LIN {X 0,Y 128.557,Z 1225.64,A -85,B 0,C 180,E1 5972.035,E2 5972.035} C_VEL
LIN {X 0,Y 143.599,Z 1214.931,A -85,B 0,C 180,E1 5965.157,E2 5965.157} C_VEL
LIN {X 0,Y 159.546,Z 1202.831,A -85,B 0,C 180,E1 5959.947,E2 5959.947} C_VEL
LIN {X 0,Y 175.745,Z 1189.232,A -85,B 0,C 180,E1 5955.959,E2 5955.959} C_VEL
LIN {X 0,Y 191.807,Z 1174.321,A -85,B 0,C 180,E1 5952.898,E2 5952.898} C_VEL
LIN {X 0,Y 207.044,Z 1158.532,A -85,B 0,C 180,E1 5950.574,E2 5950.574} C_VEL
LIN {X 0,Y 221.552,Z 1141.458,A -85,B 0,C 180,E1 5948.77,E2 5948.77} C_VEL
LIN {X 0,Y 234.912,Z 1123.521,A -85,B 0,C 180,E1 5947.392,E2 5947.392} C_VEL
LIN {X 0,Y 247.459,Z 1104.198,A -85,B 0,C 180,E1 5946.316,E2 5946.316} C_VEL
LIN {X 0,Y 258.166,Z 1084.964,A -85,B 0,C 180,E1 5945.551,E2 5945.551} C_VEL
LIN {X 0,Y 267.457,Z 1065.024,A -85,B 0,C 180,E1 5944.964,E2 5944.964} C_VEL
LIN {X 0,Y 275.777,Z 1043.211,A -85,B 0,C 180,E1 5944.432,E2 5944.432} C_VEL
LIN {X 0,Y 282.412,Z 1020.924,A -85,B 0,C 180,E1 5943.975,E2 5943.975} C_VEL
LIN {X 0,Y 287.197,Z 998.303,A -85,B 0,C 180,E1 5943.578,E2 5943.578} C_VEL
LIN {X 0,Y 291.386,Z 967,A -85,B 0,C 180,E1 5943.086,E2 5943.086} C_VEL
LIN {X 0,Y 296.698,Z 921.737,A -85,B 0,C 180,E1 5942.366,E2 5942.366} C_VEL
LIN {X 0,Y 296.244,Z 920.618,A -85,B 0,C 180,E1 5938.452,E2 5938.452} C_VEL
LIN {X 0,Y 296.574,Z 921.627,A -85,B 0,C 180,E1 5935.555,E2 5935.555} C_VEL
LIN {X 0,Y 290.553,Z 972.951,A -85,B 0,C 180,E1 5934.658,E2 5934.658} C_VEL
LIN {X 0,Y 287.245,Z 994.55,A -85,B 0,C 180,E1 5934.116,E2 5934.116} C_VEL
LIN {X 0,Y 282.043,Z 1017.129,A -85,B 0,C 180,E1 5933.394,E2 5933.394} C_VEL
LIN {X 0,Y 275.76,Z 1037.409,A -85,B 0,C 180,E1 5932.582,E2 5932.582} C_VEL
LIN {X 0,Y 267.826,Z 1057.375,A -85,B 0,C 180,E1 5931.603,E2 5931.603} C_VEL
LIN {X 0,Y 258.412,Z 1076.786,A -85,B 0,C 180,E1 5930.422,E2 5930.422} C_VEL
LIN {X 0,Y 248.14,Z 1094.686,A -85,B 0,C 180,E1 5929.083,E2 5929.083} C_VEL
LIN {X 0,Y 236.579,Z 1111.772,A -85,B 0,C 180,E1 5927.488,E2 5927.488} C_VEL
LIN {X 0,Y 224,Z 1127.849,A -85,B 0,C 180,E1 5925.599,E2 5925.599} C_VEL
LIN {X 0,Y 210.772,Z 1142.685,A -85,B 0,C 180,E1 5923.378,E2 5923.378} C_VEL
LIN {X 0,Y 196.129,Z 1156.912,A -85,B 0,C 180,E1 5920.577,E2 5920.577} C_VEL
LIN {X 0,Y 181.129,Z 1169.686,A -85,B 0,C 180,E1 5917.196,E2 5917.196} C_VEL
LIN {X 0,Y 165.996,Z 1181.07,A -85,B 0,C 180,E1 5913.054,E2 5913.054} C_VEL
LIN {X 0,Y 151.049,Z 1191.002,A -85,B 0,C 180,E1 5907.915,E2 5907.915} C_VEL
LIN {X 0,Y 136.729,Z 1199.368,A -85,B 0,C 180,E1 5901.484,E2 5901.484} C_VEL
LIN {X 0,Y 123.709,Z 1206.226,A -85,B 0,C 180,E1 5893.391,E2 5893.391} C_VEL
LIN {X 0,Y 113.281,Z 1211.302,A -85,B 0,C 180,E1 5883.783,E2 5883.783} C_VEL
LIN {X 0,Y 105.924,Z 1214.694,A -85,B 0,C 180,E1 5872.768,E2 5872.768} C_VEL
LIN {X 0,Y 102.021,Z 1216.463,A -85,B 0,C 180,E1 5861.303,E2 5861.303} C_VEL
LIN {X 0,Y 100.923,Z 1217.057,A -85,B 0,C 180,E1 5850.568,E2 5850.568} C_VEL
LIN {X 0,Y 101.896,Z 1216.542,A -85,B 0,C 180,E1 5839.255,E2 5839.255} C_VEL
LIN {X 0,Y 105.398,Z 1214.996,A -85,B 0,C 180,E1 5828.287,E2 5828.287} C_VEL
LIN {X 0,Y 112.423,Z 1211.729,A -85,B 0,C 180,E1 5817.146,E2 5817.146} C_VEL
LIN {X 0,Y 123.108,Z 1206.598,A -85,B 0,C 180,E1 5806.984,E2 5806.984} C_VEL
LIN {X 0,Y 135.387,Z 1200.239,A -85,B 0,C 180,E1 5799.157,E2 5799.157} C_VEL
LIN {X 0,Y 149.543,Z 1192.037,A -85,B 0,C 180,E1 5792.603,E2 5792.603} C_VEL
LIN {X 0,Y 164.371,Z 1182.32,A -85,B 0,C 180,E1 5787.367,E2 5787.367} C_VEL
LIN {X 0,Y 180.239,Z 1170.572,A -85,B 0,C 180,E1 5782.951,E2 5782.951} C_VEL
LIN {X 0,Y 195.213,Z 1157.984,A -85,B 0,C 180,E1 5779.542,E2 5779.542} C_VEL
LIN {X 0,Y 209.83,Z 1143.86,A -85,B 0,C 180,E1 5776.714,E2 5776.714} C_VEL
LIN {X 0,Y 223.492,Z 1128.733,A -85,B 0,C 180,E1 5774.409,E2 5774.409} C_VEL
LIN {X 0,Y 236.522,Z 1112.193,A -85,B 0,C 180,E1 5772.45,E2 5772.45} C_VEL
LIN {X 0,Y 248.371,Z 1094.704,A -85,B 0,C 180,E1 5770.817,E2 5770.817} C_VEL
LIN {X 0,Y 258.962,Z 1076.211,A -85,B 0,C 180,E1 5769.439,E2 5769.439} C_VEL
LIN {X 0,Y 268.715,Z 1055.867,A -85,B 0,C 180,E1 5768.22,E2 5768.22} C_VEL
LIN {X 0,Y 276.379,Z 1036.383,A -85,B 0,C 180,E1 5767.275,E2 5767.275} C_VEL
LIN {X 0,Y 282.83,Z 1015.172,A -85,B 0,C 180,E1 5766.44,E2 5766.44} C_VEL
LIN {X 0,Y 287.696,Z 993.438,A -85,B 0,C 180,E1 5765.758,E2 5765.758} C_VEL
LIN {X 0,Y 291.067,Z 970.64,A -85,B 0,C 180,E1 5765.196,E2 5765.196} C_VEL
LIN {X 0,Y 296.81,Z 921.706,A -85,B 0,C 180,E1 5764.329,E2 5764.329} C_VEL
LIN {X 0,Y 296.476,Z 920.939,A -85,B 0,C 180,E1 5760.773,E2 5760.773} C_VEL
LIN {X 0,Y 296.913,Z 922.137,A -85,B 0,C 180,E1 5757.598,E2 5757.598} C_VEL
LIN {X 0,Y 288.086,Z 994.765,A -85,B 0,C 180,E1 5756.486,E2 5756.486} C_VEL
LIN {X 0,Y 283.454,Z 1017.452,A -85,B 0,C 180,E1 5756.093,E2 5756.093} C_VEL
LIN {X 0,Y 277.274,Z 1039.329,A -85,B 0,C 180,E1 5755.657,E2 5755.657} C_VEL
LIN {X 0,Y 269.907,Z 1059.813,A -85,B 0,C 180,E1 5755.182,E2 5755.182} C_VEL
LIN {X 0,Y 260.611,Z 1080.49,A -85,B 0,C 180,E1 5754.602,E2 5754.602} C_VEL
LIN {X 0,Y 249.889,Z 1100.411,A -85,B 0,C 180,E1 5753.864,E2 5753.864} C_VEL
LIN {X 0,Y 238.282,Z 1118.997,A -85,B 0,C 180,E1 5752.908,E2 5752.908} C_VEL
LIN {X 0,Y 225.356,Z 1136.862,A -85,B 0,C 180,E1 5751.64,E2 5751.64} C_VEL
LIN {X 0,Y 210.819,Z 1154.455,A -85,B 0,C 180,E1 5749.924,E2 5749.924} C_VEL
LIN {X 0,Y 205.526,Z 1160.022,A -85,B 0,C 180,E1 5749.522,E2 5749.522} C_VEL
LIN {X 0,Y 190.415,Z 1173.211,A -85,B 0,C 180,E1 5749.253,E2 5749.253} C_VEL
LIN {X 0,Y 184.72,Z 1178.127,A -85,B 0,C 180,E1 5748.684,E2 5748.684} C_VEL
LIN {X 0,Y 168.259,Z 1192.432,A -85,B 0,C 180,E1 5745.598,E2 5745.598} C_VEL
LIN {X 0,Y 151.713,Z 1205.274,A -85,B 0,C 180,E1 5741.559,E2 5741.559} C_VEL
LIN {X 0,Y 134.693,Z 1217.324,A -85,B 0,C 180,E1 5735.904,E2 5735.904} C_VEL
LIN {X 0,Y 119.422,Z 1227.418,A -85,B 0,C 180,E1 5728.646,E2 5728.646} C_VEL
LIN {X 0,Y 106.632,Z 1235.615,A -85,B 0,C 180,E1 5719.419,E2 5719.419} C_VEL
LIN {X 0,Y 96.869,Z 1242.354,A -85,B 0,C 180,E1 5707.515,E2 5707.515} C_VEL
LIN {X 0,Y 91.73,Z 1247.309,A -85,B 0,C 180,E1 5693.784,E2 5693.784} C_VEL
LIN {X 0,Y 91.202,Z 1250.049,A -85,B 0,C 180,E1 5681.381,E2 5681.381} C_VEL
LIN {X 0,Y 92.698,Z 1251.177,A -85,B 0,C 180,E1 5671.854,E2 5671.854} C_VEL
LIN {X 0,Y 92.812,Z 1251.22,A -85,B 0,C 180,E1 5668.765,E2 5668.765} C_VEL
LIN {X 0,Y 91.266,Z 1250.151,A -85,B 0,C 180,E1 5659.267,E2 5659.267} C_VEL
LIN {X 0,Y 91.617,Z 1247.454,A -85,B 0,C 180,E1 5646.867,E2 5646.867} C_VEL
LIN {X 0,Y 96.53,Z 1242.58,A -85,B 0,C 180,E1 5633.077,E2 5633.077} C_VEL
LIN {X 0,Y 106.097,Z 1235.924,A -85,B 0,C 180,E1 5621.071,E2 5621.071} C_VEL
LIN {X 0,Y 118.748,Z 1227.765,A -85,B 0,C 180,E1 5611.746,E2 5611.746} C_VEL
LIN {X 0,Y 133.936,Z 1217.741,A -85,B 0,C 180,E1 5604.394,E2 5604.394} C_VEL
LIN {X 0,Y 150.911,Z 1205.757,A -85,B 0,C 180,E1 5598.663,E2 5598.663} C_VEL
LIN {X 0,Y 167.368,Z 1193.045,A -85,B 0,C 180,E1 5594.588,E2 5594.588} C_VEL
LIN {X 0,Y 183.649,Z 1178.921,A -85,B 0,C 180,E1 5591.489,E2 5591.489} C_VEL
LIN {X 0,Y 199.951,Z 1163.067,A -85,B 0,C 180,E1 5589.043,E2 5589.043} C_VEL
LIN {X 0,Y 214.685,Z 1146.942,A -85,B 0,C 180,E1 5587.261,E2 5587.261} C_VEL
LIN {X 0,Y 228.659,Z 1129.463,A -85,B 0,C 180,E1 5585.87,E2 5585.87} C_VEL
LIN {X 0,Y 241.398,Z 1111.157,A -85,B 0,C 180,E1 5584.82,E2 5584.82} C_VEL
LIN {X 0,Y 252.588,Z 1092.7,A -85,B 0,C 180,E1 5584.052,E2 5584.052} C_VEL
LIN {X 0,Y 262.931,Z 1072.464,A -85,B 0,C 180,E1 5583.45,E2 5583.45} C_VEL
LIN {X 0,Y 271.757,Z 1051.492,A -85,B 0,C 180,E1 5582.952,E2 5582.952} C_VEL
LIN {X 0,Y 279.127,Z 1029.628,A -85,B 0,C 180,E1 5582.514,E2 5582.514} C_VEL
LIN {X 0,Y 284.822,Z 1007.269,A -85,B 0,C 180,E1 5582.125,E2 5582.125} C_VEL
LIN {X 0,Y 288.68,Z 984.724,A -85,B 0,C 180,E1 5581.774,E2 5581.774} C_VEL
LIN {X 0,Y 295.41,Z 929.134,A -85,B 0,C 180,E1 5580.921,E2 5580.921} C_VEL
LIN {X 0,Y 295.275,Z 928.654,A -85,B 0,C 180,E1 5578.059,E2 5578.059} C_VEL
LIN {X 0,Y 295.326,Z 929.178,A -85,B 0,C 180,E1 5576.997,E2 5576.997} C_VEL
LIN {X 0,Y 289.639,Z 976.58,A -85,B 0,C 180,E1 5576.161,E2 5576.161} C_VEL
LIN {X 0,Y 286.245,Z 997.561,A -85,B 0,C 180,E1 5575.639,E2 5575.639} C_VEL
LIN {X 0,Y 281.067,Z 1019.164,A -85,B 0,C 180,E1 5574.966,E2 5574.966} C_VEL
LIN {X 0,Y 274.378,Z 1040.054,A -85,B 0,C 180,E1 5574.157,E2 5574.157} C_VEL
LIN {X 0,Y 266.317,Z 1059.866,A -85,B 0,C 180,E1 5573.22,E2 5573.22} C_VEL
LIN {X 0,Y 256.885,Z 1078.796,A -85,B 0,C 180,E1 5572.114,E2 5572.114} C_VEL
LIN {X 0,Y 246.122,Z 1097.056,A -85,B 0,C 180,E1 5570.803,E2 5570.803} C_VEL
LIN {X 0,Y 234.074,Z 1114.446,A -85,B 0,C 180,E1 5569.242,E2 5569.242} C_VEL
LIN {X 0,Y 220.803,Z 1130.83,A -85,B 0,C 180,E1 5567.373,E2 5567.373} C_VEL
LIN {X 0,Y 205.966,Z 1146.708,A -85,B 0,C 180,E1 5565.019,E2 5565.019} C_VEL
LIN {X 0,Y 191.033,Z 1160.637,A -85,B 0,C 180,E1 5562.279,E2 5562.279} C_VEL
LIN {X 0,Y 175.686,Z 1173.047,A -85,B 0,C 180,E1 5558.959,E2 5558.959} C_VEL
LIN {X 0,Y 160.142,Z 1184.059,A -85,B 0,C 180,E1 5554.862,E2 5554.862} C_VEL
LIN {X 0,Y 144.733,Z 1193.7,A -85,B 0,C 180,E1 5549.713,E2 5549.713} C_VEL
LIN {X 0,Y 129.906,Z 1201.869,A -85,B 0,C 180,E1 5543.172,E2 5543.172} C_VEL
LIN {X 0,Y 116.904,Z 1208.167,A -85,B 0,C 180,E1 5535.224,E2 5535.224} C_VEL
LIN {X 0,Y 105.448,Z 1213.233,A -85,B 0,C 180,E1 5524.674,E2 5524.674} C_VEL
LIN {X 0,Y 97.835,Z 1216.442,A -85,B 0,C 180,E1 5512.851,E2 5512.851} C_VEL
LIN {X 0,Y 94.04,Z 1217.965,A -85,B 0,C 180,E1 5501.033,E2 5501.033} C_VEL
LIN {X 0,Y 93.052,Z 1218.434,A -85,B 0,C 180,E1 5488.769,E2 5488.769} C_VEL
LIN {X 0,Y 94.411,Z 1217.828,A -85,B 0,C 180,E1 5477.15,E2 5477.15} C_VEL
LIN {X 0,Y 99.214,Z 1215.885,A -85,B 0,C 180,E1 5464.321,E2 5464.321} C_VEL
LIN {X 0,Y 107.616,Z 1212.43,A -85,B 0,C 180,E1 5452.851,E2 5452.851} C_VEL
LIN {X 0,Y 119.155,Z 1207.202,A -85,B 0,C 180,E1 5443.113,E2 5443.113} C_VEL
LIN {X 0,Y 133.21,Z 1200.185,A -85,B 0,C 180,E1 5435.103,E2 5435.103} C_VEL
LIN {X 0,Y 147.654,Z 1192.113,A -85,B 0,C 180,E1 5429.13,E2 5429.13} C_VEL
LIN {X 0,Y 163.284,Z 1182.136,A -85,B 0,C 180,E1 5424.166,E2 5424.166} C_VEL
LIN {X 0,Y 178.977,Z 1170.667,A -85,B 0,C 180,E1 5420.198,E2 5420.198} C_VEL
LIN {X 0,Y 194.446,Z 1157.792,A -85,B 0,C 180,E1 5416.982,E2 5416.982} C_VEL
LIN {X 0,Y 209.483,Z 1143.491,A -85,B 0,C 180,E1 5414.33,E2 5414.33} C_VEL
LIN {X 0,Y 223.024,Z 1128.54,A -85,B 0,C 180,E1 5412.231,E2 5412.231} C_VEL
LIN {X 0,Y 236.331,Z 1111.667,A -85,B 0,C 180,E1 5410.384,E2 5410.384} C_VEL
LIN {X 0,Y 247.947,Z 1094.642,A -85,B 0,C 180,E1 5408.905,E2 5408.905} C_VEL
LIN {X 0,Y 258.258,Z 1076.728,A -85,B 0,C 180,E1 5407.656,E2 5407.656} C_VEL
LIN {X 0,Y 267.702,Z 1057.251,A -85,B 0,C 180,E1 5406.551,E2 5406.551} C_VEL
LIN {X 0,Y 275.734,Z 1037.039,A -85,B 0,C 180,E1 5405.619,E2 5405.619} C_VEL
LIN {X 0,Y 282.233,Z 1015.918,A -85,B 0,C 180,E1 5404.827,E2 5404.827} C_VEL
LIN {X 0,Y 287.101,Z 994.334,A -85,B 0,C 180,E1 5404.177,E2 5404.177} C_VEL
LIN {X 0,Y 290.619,Z 970.647,A -85,B 0,C 180,E1 5403.613,E2 5403.613} C_VEL
LIN {X 0,Y 295.582,Z 929.194,A -85,B 0,C 180,E1 5402.909,E2 5402.909} C_VEL
LIN {X 0,Y 295.525,Z 929,A -85,B 0,C 180,E1 5400.194,E2 5400.194} C_VEL
LIN {X 0,Y 295.631,Z 929.49,A -85,B 0,C 180,E1 5399.038,E2 5399.038} C_VEL
LIN {X 0,Y 287.672,Z 993.536,A -85,B 0,C 180,E1 5398.096,E2 5398.096} C_VEL
LIN {X 0,Y 282.955,Z 1016.297,A -85,B 0,C 180,E1 5397.728,E2 5397.728} C_VEL
LIN {X 0,Y 276.703,Z 1038.134,A -85,B 0,C 180,E1 5397.328,E2 5397.328} C_VEL
LIN {X 0,Y 268.854,Z 1059.537,A -85,B 0,C 180,E1 5396.874,E2 5396.874} C_VEL
LIN {X 0,Y 259.481,Z 1080.086,A -85,B 0,C 180,E1 5396.353,E2 5396.353} C_VEL
LIN {X 0,Y 248.659,Z 1099.808,A -85,B 0,C 180,E1 5395.694,E2 5395.694} C_VEL
LIN {X 0,Y 236.436,Z 1118.933,A -85,B 0,C 180,E1 5394.791,E2 5394.791} C_VEL
LIN {X 0,Y 223.342,Z 1136.675,A -85,B 0,C 180,E1 5393.626,E2 5393.626} C_VEL
LIN {X 0,Y 208.955,Z 1153.639,A -85,B 0,C 180,E1 5392.085,E2 5392.085} C_VEL
LIN {X 0,Y 192.918,Z 1170.338,A -85,B 0,C 180,E1 5389.965,E2 5389.965} C_VEL
LIN {X 0,Y 184.72,Z 1178.127,A -85,B 0,C 180,E1 5388.684,E2 5388.684} C_VEL
LIN {X 0,Y 178.905,Z 1182.99,A -85,B 0,C 180,E1 5388.047,E2 5388.047} C_VEL
LIN {X 0,Y 162.487,Z 1194.342,A -85,B 0,C 180,E1 5387.224,E2 5387.224} C_VEL
LIN {X 0,Y 156.519,Z 1198.545,A -85,B 0,C 180,E1 5386.354,E2 5386.354} C_VEL
LIN {X 0,Y 139.815,Z 1210.338,A -85,B 0,C 180,E1 5382.007,E2 5382.007} C_VEL
LIN {X 0,Y 122.744,Z 1221.339,A -85,B 0,C 180,E1 5375.826,E2 5375.826} C_VEL
LIN {X 0,Y 107.622,Z 1230.478,A -85,B 0,C 180,E1 5367.715,E2 5367.715} C_VEL
LIN {X 0,Y 94.82,Z 1238.04,A -85,B 0,C 180,E1 5356.683,E2 5356.683} C_VEL
LIN {X 0,Y 86.341,Z 1243.797,A -85,B 0,C 180,E1 5342.974,E2 5342.974} C_VEL
LIN {X 0,Y 83.139,Z 1247.669,A -85,B 0,C 180,E1 5328.184,E2 5328.184} C_VEL
LIN {X 0,Y 84.079,Z 1249.483,A -85,B 0,C 180,E1 5315.459,E2 5315.459} C_VEL
LIN {X 0,Y 85.053,Z 1249.896,A -85,B 0,C 180,E1 5310,E2 5310} C_VEL
LIN {X 0,Y 83.537,Z 1249.153,A -85,B 0,C 180,E1 5301.049,E2 5301.049} C_VEL
LIN {X 0,Y 83.658,Z 1246.494,A -85,B 0,C 180,E1 5286.772,E2 5286.772} C_VEL
LIN {X 0,Y 88.842,Z 1241.894,A -85,B 0,C 180,E1 5271.759,E2 5271.759} C_VEL
LIN {X 0,Y 99.035,Z 1235.474,A -85,B 0,C 180,E1 5258.979,E2 5258.979} C_VEL
LIN {X 0,Y 112.538,Z 1227.429,A -85,B 0,C 180,E1 5249.251,E2 5249.251} C_VEL
LIN {X 0,Y 129.057,Z 1217.286,A -85,B 0,C 180,E1 5241.619,E2 5241.619} C_VEL
LIN {X 0,Y 145.817,Z 1206.162,A -85,B 0,C 180,E1 5236.272,E2 5236.272} C_VEL
LIN {X 0,Y 162.719,Z 1193.662,A -85,B 0,C 180,E1 5232.319,E2 5232.319} C_VEL
LIN {X 0,Y 179.786,Z 1179.534,A -85,B 0,C 180,E1 5229.281,E2 5229.281} C_VEL
LIN {X 0,Y 195.916,Z 1164.554,A -85,B 0,C 180,E1 5227.035,E2 5227.035} C_VEL
LIN {X 0,Y 210.884,Z 1148.771,A -85,B 0,C 180,E1 5225.354,E2 5225.354} C_VEL
LIN {X 0,Y 225.515,Z 1131.161,A -85,B 0,C 180,E1 5224.015,E2 5224.015} C_VEL
LIN {X 0,Y 238.791,Z 1112.859,A -85,B 0,C 180,E1 5223.021,E2 5223.021} C_VEL
LIN {X 0,Y 250.161,Z 1094.681,A -85,B 0,C 180,E1 5222.317,E2 5222.317} C_VEL
LIN {X 0,Y 260.581,Z 1075.111,A -85,B 0,C 180,E1 5221.779,E2 5221.779} C_VEL
LIN {X 0,Y 269.727,Z 1054.598,A -85,B 0,C 180,E1 5221.33,E2 5221.33} C_VEL
LIN {X 0,Y 277.239,Z 1033.578,A -85,B 0,C 180,E1 5220.94,E2 5220.94} C_VEL
LIN {X 0,Y 283.309,Z 1011.449,A -85,B 0,C 180,E1 5220.578,E2 5220.578} C_VEL
LIN {X 0,Y 287.781,Z 988.569,A -85,B 0,C 180,E1 5220.239,E2 5220.239} C_VEL
LIN {X 0,Y 294.301,Z 936.609,A -85,B 0,C 180,E1 5219.464,E2 5219.464} C_VEL
LIN {X 0,Y 294.278,Z 936.636,A -85,B 0,C 180,E1 5218.451,E2 5218.451} C_VEL
LIN {X 0,Y 288.807,Z 980.84,A -85,B 0,C 180,E1 5217.659,E2 5217.659} C_VEL
LIN {X 0,Y 285.183,Z 1001.957,A -85,B 0,C 180,E1 5217.133,E2 5217.133} C_VEL
LIN {X 0,Y 279.853,Z 1022.774,A -85,B 0,C 180,E1 5216.493,E2 5216.493} C_VEL
LIN {X 0,Y 272.723,Z 1043.947,A -85,B 0,C 180,E1 5215.695,E2 5215.695} C_VEL
LIN {X 0,Y 264.469,Z 1063.55,A -85,B 0,C 180,E1 5214.794,E2 5214.794} C_VEL
LIN {X 0,Y 254.492,Z 1082.794,A -85,B 0,C 180,E1 5213.703,E2 5213.703} C_VEL
LIN {X 0,Y 243.09,Z 1101.272,A -85,B 0,C 180,E1 5212.407,E2 5212.407} C_VEL
LIN {X 0,Y 230.855,Z 1118.27,A -85,B 0,C 180,E1 5210.918,E2 5210.918} C_VEL
LIN {X 0,Y 217.326,Z 1134.38,A -85,B 0,C 180,E1 5209.127,E2 5209.127} C_VEL
LIN {X 0,Y 203.154,Z 1148.982,A -85,B 0,C 180,E1 5207.023,E2 5207.023} C_VEL
LIN {X 0,Y 187.88,Z 1162.761,A -85,B 0,C 180,E1 5204.411,E2 5204.411} C_VEL
LIN {X 0,Y 172.134,Z 1175.102,A -85,B 0,C 180,E1 5201.222,E2 5201.222} C_VEL
LIN {X 0,Y 156.104,Z 1185.993,A -85,B 0,C 180,E1 5197.265,E2 5197.265} C_VEL
LIN {X 0,Y 139.336,Z 1195.94,A -85,B 0,C 180,E1 5191.958,E2 5191.958} C_VEL
LIN {X 0,Y 124.592,Z 1203.634,A -85,B 0,C 180,E1 5185.747,E2 5185.747} C_VEL
LIN {X 0,Y 110.233,Z 1210.107,A -85,B 0,C 180,E1 5177.28,E2 5177.28} C_VEL
LIN {X 0,Y 98.418,Z 1214.863,A -85,B 0,C 180,E1 5166.621,E2 5166.621} C_VEL
LIN {X 0,Y 90.287,Z 1217.932,A -85,B 0,C 180,E1 5154.188,E2 5154.188} C_VEL
LIN {X 0,Y 86.303,Z 1219.359,A -85,B 0,C 180,E1 5142.036,E2 5142.036} C_VEL
LIN {X 0,Y 85.175,Z 1219.824,A -85,B 0,C 180,E1 5128.655,E2 5128.655} C_VEL
LIN {X 0,Y 86.725,Z 1219.222,A -85,B 0,C 180,E1 5115.989,E2 5115.989} C_VEL
LIN {X 0,Y 92.124,Z 1217.285,A -85,B 0,C 180,E1 5102.181,E2 5102.181} C_VEL
LIN {X 0,Y 101.385,Z 1213.834,A -85,B 0,C 180,E1 5090.133,E2 5090.133} C_VEL
LIN {X 0,Y 113.86,Z 1208.606,A -85,B 0,C 180,E1 5080.185,E2 5080.185} C_VEL
LIN {X 0,Y 128.793,Z 1201.59,A -85,B 0,C 180,E1 5072.203,E2 5072.203} C_VEL
LIN {X 0,Y 143.946,Z 1193.516,A -85,B 0,C 180,E1 5066.361,E2 5066.361} C_VEL
LIN {X 0,Y 160.193,Z 1183.538,A -85,B 0,C 180,E1 5061.57,E2 5061.57} C_VEL
LIN {X 0,Y 176.393,Z 1172.066,A -85,B 0,C 180,E1 5057.777,E2 5057.777} C_VEL
LIN {X 0,Y 192.281,Z 1159.189,A -85,B 0,C 180,E1 5054.722,E2 5054.722} C_VEL
LIN {X 0,Y 207.665,Z 1144.885,A -85,B 0,C 180,E1 5052.213,E2 5052.213} C_VEL
LIN {X 0,Y 221.95,Z 1129.404,A -85,B 0,C 180,E1 5050.171,E2 5050.171} C_VEL
LIN {X 0,Y 235.506,Z 1112.417,A -85,B 0,C 180,E1 5048.433,E2 5048.433} C_VEL
LIN {X 0,Y 247.322,Z 1095.25,A -85,B 0,C 180,E1 5047.041,E2 5047.041} C_VEL
LIN {X 0,Y 257.806,Z 1077.246,A -85,B 0,C 180,E1 5045.866,E2 5045.866} C_VEL
LIN {X 0,Y 267.399,Z 1057.54,A -85,B 0,C 180,E1 5044.818,E2 5044.818} C_VEL
LIN {X 0,Y 275.32,Z 1037.687,A -85,B 0,C 180,E1 5043.957,E2 5043.957} C_VEL
LIN {X 0,Y 281.877,Z 1016.611,A -85,B 0,C 180,E1 5043.206,E2 5043.206} C_VEL
LIN {X 0,Y 286.743,Z 995.142,A -85,B 0,C 180,E1 5042.589,E2 5042.589} C_VEL
LIN {X 0,Y 290.512,Z 969.67,A -85,B 0,C 180,E1 5042.007,E2 5042.007} C_VEL
LIN {X 0,Y 294.523,Z 936.791,A -85,B 0,C 180,E1 5041.459,E2 5041.459} C_VEL
LIN {X 0,Y 294.509,Z 937.085,A -85,B 0,C 180,E1 5040.487,E2 5040.487} C_VEL
LIN {X 0,Y 287.454,Z 992.467,A -85,B 0,C 180,E1 5039.707,E2 5039.707} C_VEL
LIN {X 0,Y 282.687,Z 1015.142,A -85,B 0,C 180,E1 5039.367,E2 5039.367} C_VEL
LIN {X 0,Y 276.245,Z 1037.312,A -85,B 0,C 180,E1 5038.997,E2 5038.997} C_VEL
LIN {X 0,Y 268.533,Z 1058.112,A -85,B 0,C 180,E1 5038.602,E2 5038.602} C_VEL
LIN {X 0,Y 259.091,Z 1078.661,A -85,B 0,C 180,E1 5038.143,E2 5038.143} C_VEL
LIN {X 0,Y 248.181,Z 1098.377,A -85,B 0,C 180,E1 5037.568,E2 5037.568} C_VEL
LIN {X 0,Y 235.877,Z 1117.433,A -85,B 0,C 180,E1 5036.774,E2 5036.774} C_VEL
LIN {X 0,Y 222.579,Z 1135.227,A -85,B 0,C 180,E1 5035.731,E2 5035.731} C_VEL
LIN {X 0,Y 207.978,Z 1152.183,A -85,B 0,C 180,E1 5034.341,E2 5034.341} C_VEL
LIN {X 0,Y 191.644,Z 1168.873,A -85,B 0,C 180,E1 5032.414,E2 5032.414} C_VEL
LIN {X 0,Y 175.613,Z 1183.376,A -85,B 0,C 180,E1 5030.047,E2 5030.047} C_VEL
LIN {X 0,Y 159.1,Z 1196.558,A -85,B 0,C 180,E1 5026.922,E2 5026.922} C_VEL
LIN {X 0,Y 156.519,Z 1198.545,A -85,B 0,C 180,E1 5026.354,E2 5026.354} C_VEL
LIN {X 0,Y 150.469,Z 1202.656,A -85,B 0,C 180,E1 5025.377,E2 5025.377} C_VEL
LIN {X 0,Y 133.145,Z 1212.032,A -85,B 0,C 180,E1 5023.627,E2 5023.627} C_VEL
LIN {X 0,Y 126.976,Z 1215.409,A -85,B 0,C 180,E1 5022.213,E2 5022.213} C_VEL
LIN {X 0,Y 109.263,Z 1225.679,A -85,B 0,C 180,E1 5014.946,E2 5014.946} C_VEL
LIN {X 0,Y 94.585,Z 1233.716,A -85,B 0,C 180,E1 5005.539,E2 5005.539} C_VEL
LIN {X 0,Y 82.837,Z 1240.19,A -85,B 0,C 180,E1 4992.525,E2 4992.525} C_VEL
LIN {X 0,Y 76.258,Z 1244.884,A -85,B 0,C 180,E1 4976.473,E2 4976.473} C_VEL
LIN {X 0,Y 75.416,Z 1247.622,A -85,B 0,C 180,E1 4960.696,E2 4960.696} C_VEL
LIN {X 0,Y 77.147,Z 1248.5,A -85,B 0,C 180,E1 4950,E2 4950} C_VEL
LIN {X 0,Y 75.349,Z 1247.493,A -85,B 0,C 180,E1 4938.519,E2 4938.519} C_VEL
LIN {X 0,Y 76.259,Z 1244.86,A -85,B 0,C 180,E1 4923.527,E2 4923.527} C_VEL
LIN {X 0,Y 83.272,Z 1239.882,A -85,B 0,C 180,E1 4906.813,E2 4906.813} C_VEL
LIN {X 0,Y 95.218,Z 1233.308,A -85,B 0,C 180,E1 4893.949,E2 4893.949} C_VEL
LIN {X 0,Y 110.793,Z 1224.78,A -85,B 0,C 180,E1 4884.293,E2 4884.293} C_VEL
LIN {X 0,Y 127.886,Z 1214.756,A -85,B 0,C 180,E1 4877.482,E2 4877.482} C_VEL
LIN {X 0,Y 146.398,Z 1202.785,A -85,B 0,C 180,E1 4872.413,E2 4872.413} C_VEL
LIN {X 0,Y 163.948,Z 1190.081,A -85,B 0,C 180,E1 4868.905,E2 4868.905} C_VEL
LIN {X 0,Y 181.065,Z 1175.971,A -85,B 0,C 180,E1 4866.307,E2 4866.307} C_VEL
LIN {X 0,Y 198.021,Z 1160.13,A -85,B 0,C 180,E1 4864.291,E2 4864.291} C_VEL
LIN {X 0,Y 213.72,Z 1143.441,A -85,B 0,C 180,E1 4862.81,E2 4862.81} C_VEL
LIN {X 0,Y 228.063,Z 1125.925,A -85,B 0,C 180,E1 4861.715,E2 4861.715} C_VEL
LIN {X 0,Y 240.989,Z 1107.638,A -85,B 0,C 180,E1 4860.913,E2 4860.913} C_VEL
LIN {X 0,Y 252.96,Z 1087.985,A -85,B 0,C 180,E1 4860.314,E2 4860.314} C_VEL
LIN {X 0,Y 263.455,Z 1067.546,A -85,B 0,C 180,E1 4859.873,E2 4859.873} C_VEL
LIN {X 0,Y 271.963,Z 1047.163,A -85,B 0,C 180,E1 4859.505,E2 4859.505} C_VEL
LIN {X 0,Y 279.639,Z 1024.105,A -85,B 0,C 180,E1 4859.142,E2 4859.142} C_VEL
LIN {X 0,Y 285.183,Z 1001.927,A -85,B 0,C 180,E1 4858.825,E2 4858.825} C_VEL
LIN {X 0,Y 285.473,Z 1000.409,A -85,B 0,C 180,E1 4858.795,E2 4858.795} C_VEL
LIN {X 0,Y 280.124,Z 1021.966,A -85,B 0,C 180,E1 4858.179,E2 4858.179} C_VEL
LIN {X 0,Y 273.224,Z 1042.85,A -85,B 0,C 180,E1 4857.446,E2 4857.446} C_VEL
LIN {X 0,Y 264.919,Z 1062.66,A -85,B 0,C 180,E1 4856.605,E2 4856.605} C_VEL
LIN {X 0,Y 255.201,Z 1081.588,A -85,B 0,C 180,E1 4855.621,E2 4855.621} C_VEL
LIN {X 0,Y 244.098,Z 1099.848,A -85,B 0,C 180,E1 4854.46,E2 4854.46} C_VEL
LIN {X 0,Y 231.647,Z 1117.24,A -85,B 0,C 180,E1 4853.081,E2 4853.081} C_VEL
LIN {X 0,Y 217.894,Z 1133.626,A -85,B 0,C 180,E1 4851.432,E2 4851.432} C_VEL
LIN {X 0,Y 202.452,Z 1149.507,A -85,B 0,C 180,E1 4849.351,E2 4849.351} C_VEL
LIN {X 0,Y 186.818,Z 1163.44,A -85,B 0,C 180,E1 4846.917,E2 4846.917} C_VEL
LIN {X 0,Y 170.628,Z 1175.854,A -85,B 0,C 180,E1 4843.943,E2 4843.943} C_VEL
LIN {X 0,Y 154.061,Z 1186.869,A -85,B 0,C 180,E1 4840.224,E2 4840.224} C_VEL
LIN {X 0,Y 137.392,Z 1196.513,A -85,B 0,C 180,E1 4835.457,E2 4835.457} C_VEL
LIN {X 0,Y 120.837,Z 1204.777,A -85,B 0,C 180,E1 4829.134,E2 4829.134} C_VEL
LIN {X 0,Y 106.291,Z 1210.978,A -85,B 0,C 180,E1 4821.329,E2 4821.329} C_VEL
LIN {X 0,Y 92.81,Z 1216.041,A -85,B 0,C 180,E1 4810.268,E2 4810.268} C_VEL
LIN {X 0,Y 83.447,Z 1219.242,A -85,B 0,C 180,E1 4797.084,E2 4797.084} C_VEL
LIN {X 0,Y 78.599,Z 1220.752,A -85,B 0,C 180,E1 4783.237,E2 4783.237} C_VEL
LIN {X 0,Y 77.298,Z 1221.214,A -85,B 0,C 180,E1 4768.518,E2 4768.518} C_VEL
LIN {X 0,Y 78.907,Z 1220.669,A -85,B 0,C 180,E1 4755.32,E2 4755.32} C_VEL
LIN {X 0,Y 84.455,Z 1218.952,A -85,B 0,C 180,E1 4740.962,E2 4740.962} C_VEL
LIN {X 0,Y 94.33,Z 1215.588,A -85,B 0,C 180,E1 4728.106,E2 4728.106} C_VEL
LIN {X 0,Y 107.551,Z 1210.545,A -85,B 0,C 180,E1 4717.797,E2 4717.797} C_VEL
LIN {X 0,Y 123.213,Z 1203.724,A -85,B 0,C 180,E1 4709.742,E2 4709.742} C_VEL
LIN {X 0,Y 139.775,Z 1195.391,A -85,B 0,C 180,E1 4703.709,E2 4703.709} C_VEL
LIN {X 0,Y 156.58,Z 1185.468,A -85,B 0,C 180,E1 4699.084,E2 4699.084} C_VEL
LIN {X 0,Y 173.24,Z 1174.118,A -85,B 0,C 180,E1 4695.461,E2 4695.461} C_VEL
LIN {X 0,Y 189.506,Z 1161.38,A -85,B 0,C 180,E1 4692.564,E2 4692.564} C_VEL
LIN {X 0,Y 205.203,Z 1147.168,A -85,B 0,C 180,E1 4690.191,E2 4690.191} C_VEL
LIN {X 0,Y 219.273,Z 1132.38,A -85,B 0,C 180,E1 4688.325,E2 4688.325} C_VEL
LIN {X 0,Y 233.456,Z 1115.174,A -85,B 0,C 180,E1 4686.641,E2 4686.641} C_VEL
LIN {X 0,Y 245.517,Z 1098.16,A -85,B 0,C 180,E1 4685.324,E2 4685.324} C_VEL
LIN {X 0,Y 256.1,Z 1080.454,A -85,B 0,C 180,E1 4684.219,E2 4684.219} C_VEL
LIN {X 0,Y 266.364,Z 1060.019,A -85,B 0,C 180,E1 4683.181,E2 4683.181} C_VEL
LIN {X 0,Y 274.437,Z 1040.394,A -85,B 0,C 180,E1 4682.367,E2 4682.367} C_VEL
LIN {X 0,Y 281.218,Z 1019.119,A -85,B 0,C 180,E1 4681.639,E2 4681.639} C_VEL
LIN {X 0,Y 285.307,Z 1002.632,A -85,B 0,C 180,E1 4681.166,E2 4681.166} C_VEL
LIN {X 0,Y 279.669,Z 1024.882,A -85,B 0,C 180,E1 4680.848,E2 4680.848} C_VEL
LIN {X 0,Y 272.464,Z 1046.51,A -85,B 0,C 180,E1 4680.508,E2 4680.508} C_VEL
LIN {X 0,Y 263.955,Z 1067.009,A -85,B 0,C 180,E1 4680.142,E2 4680.142} C_VEL
LIN {X 0,Y 253.632,Z 1087.191,A -85,B 0,C 180,E1 4679.711,E2 4679.711} C_VEL
LIN {X 0,Y 241.487,Z 1107.238,A -85,B 0,C 180,E1 4679.109,E2 4679.109} C_VEL
LIN {X 0,Y 228.56,Z 1125.586,A -85,B 0,C 180,E1 4678.313,E2 4678.313} C_VEL
LIN {X 0,Y 214.214,Z 1143.124,A -85,B 0,C 180,E1 4677.225,E2 4677.225} C_VEL
LIN {X 0,Y 198.51,Z 1159.854,A -85,B 0,C 180,E1 4675.755,E2 4675.755} C_VEL
LIN {X 0,Y 182.028,Z 1175.32,A -85,B 0,C 180,E1 4673.816,E2 4673.816} C_VEL
LIN {X 0,Y 164.89,Z 1189.477,A -85,B 0,C 180,E1 4671.252,E2 4671.252} C_VEL
LIN {X 0,Y 147.307,Z 1202.276,A -85,B 0,C 180,E1 4667.79,E2 4667.79} C_VEL
LIN {X 0,Y 128.741,Z 1214.334,A -85,B 0,C 180,E1 4662.792,E2 4662.792} C_VEL
LIN {X 0,Y 126.976,Z 1215.409,A -85,B 0,C 180,E1 4662.213,E2 4662.213} C_VEL
LIN {X 0,Y 120.834,Z 1218.732,A -85,B 0,C 180,E1 4660.623,E2 4660.623} C_VEL
LIN {X 0,Y 103.342,Z 1225.994,A -85,B 0,C 180,E1 4657.127,E2 4657.127} C_VEL
LIN {X 0,Y 97.373,Z 1228.581,A -85,B 0,C 180,E1 4654.707,E2 4654.707} C_VEL
LIN {X 0,Y 82.323,Z 1236.011,A -85,B 0,C 180,E1 4643.282,E2 4643.282} C_VEL
LIN {X 0,Y 71.75,Z 1241.498,A -85,B 0,C 180,E1 4627.817,E2 4627.817} C_VEL
LIN {X 0,Y 67.342,Z 1245.232,A -85,B 0,C 180,E1 4609.065,E2 4609.065} C_VEL
LIN {X 0,Y 68.383,Z 1246.817,A -85,B 0,C 180,E1 4594.192,E2 4594.192} C_VEL
LIN {X 0,Y 69.168,Z 1247.092,A -85,B 0,C 180,E1 4590,E2 4590} C_VEL
LIN {X 0,Y 67.308,Z 1245.932,A -85,B 0,C 180,E1 4576.251,E2 4576.251} C_VEL
LIN {X 0,Y 69.372,Z 1243.051,A -85,B 0,C 180,E1 4558.745,E2 4558.745} C_VEL
LIN {X 0,Y 77.873,Z 1238.132,A -85,B 0,C 180,E1 4541.869,E2 4541.869} C_VEL
LIN {X 0,Y 91.478,Z 1231.453,A -85,B 0,C 180,E1 4529.028,E2 4529.028} C_VEL
LIN {X 0,Y 107.92,Z 1223.123,A -85,B 0,C 180,E1 4520.046,E2 4520.046} C_VEL
LIN {X 0,Y 125.609,Z 1213.266,A -85,B 0,C 180,E1 4513.809,E2 4513.809} C_VEL
LIN {X 0,Y 145.006,Z 1201.175,A -85,B 0,C 180,E1 4509.124,E2 4509.124} C_VEL
LIN {X 0,Y 162.861,Z 1188.599,A -85,B 0,C 180,E1 4505.99,E2 4505.99} C_VEL
LIN {X 0,Y 180.339,Z 1174.497,A -85,B 0,C 180,E1 4503.672,E2 4503.672} C_VEL
LIN {X 0,Y 197.573,Z 1158.663,A -85,B 0,C 180,E1 4501.891,E2 4501.891} C_VEL
LIN {X 0,Y 213.291,Z 1142.195,A -85,B 0,C 180,E1 4500.612,E2 4500.612} C_VEL
LIN {X 0,Y 227.965,Z 1124.473,A -85,B 0,C 180,E1 4499.653,E2 4499.653} C_VEL
LIN {X 0,Y 240.997,Z 1106.193,A -85,B 0,C 180,E1 4498.972,E2 4498.972} C_VEL
LIN {X 0,Y 253.046,Z 1086.545,A -85,B 0,C 180,E1 4498.474,E2 4498.474} C_VEL
LIN {X 0,Y 262.581,Z 1068.165,A -85,B 0,C 180,E1 4498.124,E2 4498.124} C_VEL
LIN {X 0,Y 252.268,Z 1087.319,A -85,B 0,C 180,E1 4497.154,E2 4497.154} C_VEL
LIN {X 0,Y 240.538,Z 1105.473,A -85,B 0,C 180,E1 4496.022,E2 4496.022} C_VEL
LIN {X 0,Y 226.961,Z 1123.386,A -85,B 0,C 180,E1 4494.62,E2 4494.62} C_VEL
LIN {X 0,Y 213.225,Z 1139.012,A -85,B 0,C 180,E1 4493.068,E2 4493.068} C_VEL
LIN {X 0,Y 198.306,Z 1153.529,A -85,B 0,C 180,E1 4491.19,E2 4491.19} C_VEL
LIN {X 0,Y 182.394,Z 1167.008,A -85,B 0,C 180,E1 4488.879,E2 4488.879} C_VEL
LIN {X 0,Y 165.883,Z 1179.179,A -85,B 0,C 180,E1 4486.024,E2 4486.024} C_VEL
LIN {X 0,Y 148.696,Z 1189.991,A -85,B 0,C 180,E1 4482.386,E2 4482.386} C_VEL
LIN {X 0,Y 131.133,Z 1199.483,A -85,B 0,C 180,E1 4477.589,E2 4477.589} C_VEL
LIN {X 0,Y 114.039,Z 1207.398,A -85,B 0,C 180,E1 4471.252,E2 4471.252} C_VEL
LIN {X 0,Y 98.071,Z 1213.714,A -85,B 0,C 180,E1 4462.674,E2 4462.674} C_VEL
LIN {X 0,Y 84.7,Z 1218.149,A -85,B 0,C 180,E1 4451.38,E2 4451.38} C_VEL
LIN {X 0,Y 74.804,Z 1221.067,A -85,B 0,C 180,E1 4436.418,E2 4436.418} C_VEL
LIN {X 0,Y 70.169,Z 1222.421,A -85,B 0,C 180,E1 4420.507,E2 4420.507} C_VEL
LIN {X 0,Y 69.504,Z 1222.549,A -85,B 0,C 180,E1 4405.875,E2 4405.875} C_VEL
LIN {X 0,Y 72.161,Z 1221.857,A -85,B 0,C 180,E1 4390.577,E2 4390.577} C_VEL
LIN {X 0,Y 79.28,Z 1219.823,A -85,B 0,C 180,E1 4375.423,E2 4375.423} C_VEL
LIN {X 0,Y 90.345,Z 1216.446,A -85,B 0,C 180,E1 4363.08,E2 4363.08} C_VEL
LIN {X 0,Y 105.014,Z 1211.15,A -85,B 0,C 180,E1 4353.087,E2 4353.087} C_VEL
LIN {X 0,Y 121.054,Z 1204.4,A -85,B 0,C 180,E1 4345.806,E2 4345.806} C_VEL
LIN {X 0,Y 137.618,Z 1196.323,A -85,B 0,C 180,E1 4340.411,E2 4340.411} C_VEL
LIN {X 0,Y 155.052,Z 1186.342,A -85,B 0,C 180,E1 4336.096,E2 4336.096} C_VEL
LIN {X 0,Y 172.21,Z 1174.864,A -85,B 0,C 180,E1 4332.739,E2 4332.739} C_VEL
LIN {X 0,Y 188.926,Z 1161.938,A -85,B 0,C 180,E1 4330.059,E2 4330.059} C_VEL
LIN {X 0,Y 204.901,Z 1147.673,A -85,B 0,C 180,E1 4327.883,E2 4327.883} C_VEL
LIN {X 0,Y 219.711,Z 1132.186,A -85,B 0,C 180,E1 4326.111,E2 4326.111} C_VEL
LIN {X 0,Y 233.713,Z 1115.195,A -85,B 0,C 180,E1 4324.602,E2 4324.602} C_VEL
LIN {X 0,Y 245.888,Z 1098.023,A -85,B 0,C 180,E1 4323.39,E2 4323.39} C_VEL
LIN {X 0,Y 256.674,Z 1080.017,A -85,B 0,C 180,E1 4322.363,E2 4322.363} C_VEL
LIN {X 0,Y 262.221,Z 1069.415,A -85,B 0,C 180,E1 4321.843,E2 4321.843} C_VEL
LIN {X 0,Y 251.538,Z 1089.716,A -85,B 0,C 180,E1 4321.461,E2 4321.461} C_VEL
LIN {X 0,Y 239.647,Z 1108.586,A -85,B 0,C 180,E1 4320.957,E2 4320.957} C_VEL
LIN {X 0,Y 225.963,Z 1127.29,A -85,B 0,C 180,E1 4320.221,E2 4320.221} C_VEL
LIN {X 0,Y 211.482,Z 1144.5,A -85,B 0,C 180,E1 4319.248,E2 4319.248} C_VEL
LIN {X 0,Y 195.965,Z 1160.467,A -85,B 0,C 180,E1 4317.954,E2 4317.954} C_VEL
LIN {X 0,Y 178.927,Z 1175.863,A -85,B 0,C 180,E1 4316.156,E2 4316.156} C_VEL
LIN {X 0,Y 161.902,Z 1189.457,A -85,B 0,C 180,E1 4313.857,E2 4313.857} C_VEL
LIN {X 0,Y 143.89,Z 1202.054,A -85,B 0,C 180,E1 4310.644,E2 4310.644} C_VEL
LIN {X 0,Y 125.59,Z 1213.376,A -85,B 0,C 180,E1 4306.183,E2 4306.183} C_VEL
LIN {X 0,Y 107.594,Z 1223.362,A -85,B 0,C 180,E1 4299.809,E2 4299.809} C_VEL
LIN {X 0,Y 97.373,Z 1228.581,A -85,B 0,C 180,E1 4294.707,E2 4294.707} C_VEL
LIN {X 0,Y 91.555,Z 1231.052,A -85,B 0,C 180,E1 4291.935,E2 4291.935} C_VEL
LIN {X 0,Y 74.721,Z 1236.131,A -85,B 0,C 180,E1 4284.371,E2 4284.371} C_VEL
LIN {X 0,Y 70.172,Z 1237.789,A -85,B 0,C 180,E1 4280.153,E2 4280.153} C_VEL
LIN {X 0,Y 61.272,Z 1242.287,A -85,B 0,C 180,E1 4261.478,E2 4261.478} C_VEL
LIN {X 0,Y 59.578,Z 1244.978,A -85,B 0,C 180,E1 4240.638,E2 4240.638} C_VEL
LIN {X 0,Y 61.162,Z 1245.679,A -85,B 0,C 180,E1 4230,E2 4230} C_VEL
LIN {X 0,Y 59.359,Z 1244.362,A -85,B 0,C 180,E1 4213.361,E2 4213.361} C_VEL
LIN {X 0,Y 62.708,Z 1241.407,A -85,B 0,C 180,E1 4193.848,E2 4193.848} C_VEL
LIN {X 0,Y 73.125,Z 1236.379,A -85,B 0,C 180,E1 4176.226,E2 4176.226} C_VEL
LIN {X 0,Y 88.463,Z 1229.598,A -85,B 0,C 180,E1 4163.726,E2 4163.726} C_VEL
LIN {X 0,Y 106.717,Z 1220.962,A -85,B 0,C 180,E1 4155.204,E2 4155.204} C_VEL
LIN {X 0,Y 125.725,Z 1210.741,A -85,B 0,C 180,E1 4149.562,E2 4149.562} C_VEL
LIN {X 0,Y 144.686,Z 1199.182,A -85,B 0,C 180,E1 4145.681,E2 4145.681} C_VEL
LIN {X 0,Y 163.184,Z 1186.364,A -85,B 0,C 180,E1 4142.919,E2 4142.919} C_VEL
LIN {X 0,Y 180.992,Z 1172.202,A -85,B 0,C 180,E1 4140.926,E2 4140.926} C_VEL
LIN {X 0,Y 197.975,Z 1156.712,A -85,B 0,C 180,E1 4139.45,E2 4139.45} C_VEL
LIN {X 0,Y 214.051,Z 1139.947,A -85,B 0,C 180,E1 4138.357,E2 4138.357} C_VEL
LIN {X 0,Y 228.805,Z 1122.221,A -85,B 0,C 180,E1 4137.565,E2 4137.565} C_VEL
LIN {X 0,Y 233.964,Z 1115.244,A -85,B 0,C 180,E1 4137.336,E2 4137.336} C_VEL
LIN {X 0,Y 220.493,Z 1131.668,A -85,B 0,C 180,E1 4136.022,E2 4136.022} C_VEL
LIN {X 0,Y 205.921,Z 1146.852,A -85,B 0,C 180,E1 4134.474,E2 4134.474} C_VEL
LIN {X 0,Y 189.589,Z 1161.533,A -85,B 0,C 180,E1 4132.501,E2 4132.501} C_VEL
LIN {X 0,Y 172.547,Z 1174.742,A -85,B 0,C 180,E1 4130.086,E2 4130.086} C_VEL
LIN {X 0,Y 154.913,Z 1186.472,A -85,B 0,C 180,E1 4127.051,E2 4127.051} C_VEL
LIN {X 0,Y 137.746,Z 1196.15,A -85,B 0,C 180,E1 4123.359,E2 4123.359} C_VEL
LIN {X 0,Y 118.691,Z 1205.309,A -85,B 0,C 180,E1 4117.913,E2 4117.913} C_VEL
LIN {X 0,Y 101.709,Z 1212.191,A -85,B 0,C 180,E1 4111.033,E2 4111.033} C_VEL
LIN {X 0,Y 85.806,Z 1217.547,A -85,B 0,C 180,E1 4101.324,E2 4101.324} C_VEL
LIN {X 0,Y 72.917,Z 1221.168,A -85,B 0,C 180,E1 4088.1,E2 4088.1} C_VEL
LIN {X 0,Y 64.501,Z 1223.279,A -85,B 0,C 180,E1 4070.887,E2 4070.887} C_VEL
LIN {X 0,Y 61.647,Z 1223.932,A -85,B 0,C 180,E1 4054.651,E2 4054.651} C_VEL
LIN {X 0,Y 62.448,Z 1223.821,A -85,B 0,C 180,E1 4037.987,E2 4037.987} C_VEL
LIN {X 0,Y 67.875,Z 1222.481,A -85,B 0,C 180,E1 4020.36,E2 4020.36} C_VEL
LIN {X 0,Y 78.87,Z 1219.622,A -85,B 0,C 180,E1 4004.773,E2 4004.773} C_VEL
LIN {X 0,Y 93.407,Z 1215.209,A -85,B 0,C 180,E1 3993.394,E2 3993.394} C_VEL
LIN {X 0,Y 109.565,Z 1209.235,A -85,B 0,C 180,E1 3985.389,E2 3985.389} C_VEL
LIN {X 0,Y 127.87,Z 1201.226,A -85,B 0,C 180,E1 3979.173,E2 3979.173} C_VEL
LIN {X 0,Y 145.767,Z 1191.971,A -85,B 0,C 180,E1 3974.731,E2 3974.731} C_VEL
LIN {X 0,Y 163.177,Z 1181.367,A -85,B 0,C 180,E1 3971.375,E2 3971.375} C_VEL
LIN {X 0,Y 180.052,Z 1169.365,A -85,B 0,C 180,E1 3968.724,E2 3968.724} C_VEL
LIN {X 0,Y 196.262,Z 1156.078,A -85,B 0,C 180,E1 3966.588,E2 3966.588} C_VEL
LIN {X 0,Y 211.711,Z 1141.388,A -85,B 0,C 180,E1 3964.816,E2 3964.816} C_VEL
LIN {X 0,Y 225.851,Z 1125.716,A -85,B 0,C 180,E1 3963.369,E2 3963.369} C_VEL
LIN {X 0,Y 233.469,Z 1116.251,A -85,B 0,C 180,E1 3962.644,E2 3962.644} C_VEL
LIN {X 0,Y 219.086,Z 1134.454,A -85,B 0,C 180,E1 3961.924,E2 3961.924} C_VEL
LIN {X 0,Y 203.994,Z 1150.998,A -85,B 0,C 180,E1 3960.979,E2 3960.979} C_VEL
LIN {X 0,Y 187.759,Z 1166.46,A -85,B 0,C 180,E1 3959.695,E2 3959.695} C_VEL
LIN {X 0,Y 170.084,Z 1181.248,A -85,B 0,C 180,E1 3957.91,E2 3957.91} C_VEL
LIN {X 0,Y 151.457,Z 1194.883,A -85,B 0,C 180,E1 3955.42,E2 3955.42} C_VEL
LIN {X 0,Y 132.286,Z 1207.026,A -85,B 0,C 180,E1 3951.934,E2 3951.934} C_VEL
LIN {X 0,Y 112.925,Z 1217.804,A -85,B 0,C 180,E1 3946.889,E2 3946.889} C_VEL
LIN {X 0,Y 94.843,Z 1226.745,A -85,B 0,C 180,E1 3939.756,E2 3939.756} C_VEL
LIN {X 0,Y 78.25,Z 1234.208,A -85,B 0,C 180,E1 3928.88,E2 3928.88} C_VEL
LIN {X 0,Y 70.172,Z 1237.789,A -85,B 0,C 180,E1 3920.153,E2 3920.153} C_VEL
LIN {X 0,Y 65.683,Z 1239.407,A -85,B 0,C 180,E1 3914.988,E2 3914.988} C_VEL
LIN {X 0,Y 53.045,Z 1242.095,A -85,B 0,C 180,E1 3897.816,E2 3897.816} C_VEL
LIN {X 0,Y 51.625,Z 1242.707,A -85,B 0,C 180,E1 3891.316,E2 3891.316} C_VEL
LIN {X 0,Y 52.995,Z 1244.232,A -85,B 0,C 180,E1 3870.711,E2 3870.711} C_VEL
LIN {X 0,Y 52.38,Z 1244.016,A -85,B 0,C 180,E1 3865.621,E2 3865.621} C_VEL
LIN {X 0,Y 51.985,Z 1242.297,A -85,B 0,C 180,E1 3844.968,E2 3844.968} C_VEL
LIN {X 0,Y 59.405,Z 1238.504,A -85,B 0,C 180,E1 3822.221,E2 3822.221} C_VEL
LIN {X 0,Y 73.492,Z 1232.98,A -85,B 0,C 180,E1 3806.116,E2 3806.116} C_VEL
LIN {X 0,Y 91.388,Z 1225.555,A -85,B 0,C 180,E1 3795.685,E2 3795.685} C_VEL
LIN {X 0,Y 110.378,Z 1216.688,A -85,B 0,C 180,E1 3789.124,E2 3789.124} C_VEL
LIN {X 0,Y 130.398,Z 1205.995,A -85,B 0,C 180,E1 3784.602,E2 3784.602} C_VEL
LIN {X 0,Y 150.055,Z 1193.905,A -85,B 0,C 180,E1 3781.527,E2 3781.527} C_VEL
LIN {X 0,Y 168.981,Z 1180.365,A -85,B 0,C 180,E1 3779.371,E2 3779.371} C_VEL
LIN {X 0,Y 187.103,Z 1165.496,A -85,B 0,C 180,E1 3777.823,E2 3777.823} C_VEL
LIN {X 0,Y 203.798,Z 1149.819,A -85,B 0,C 180,E1 3776.725,E2 3776.725} C_VEL
LIN {X 0,Y 205.04,Z 1148.516,A -85,B 0,C 180,E1 3776.645,E2 3776.645} C_VEL
LIN {X 0,Y 188.719,Z 1162.933,A -85,B 0,C 180,E1 3774.886,E2 3774.886} C_VEL
LIN {X 0,Y 171.36,Z 1176.144,A -85,B 0,C 180,E1 3772.7,E2 3772.7} C_VEL
LIN {X 0,Y 153.328,Z 1187.876,A -85,B 0,C 180,E1 3769.946,E2 3769.946} C_VEL
LIN {X 0,Y 135.681,Z 1197.556,A -85,B 0,C 180,E1 3766.581,E2 3766.581} C_VEL
LIN {X 0,Y 115.932,Z 1206.715,A -85,B 0,C 180,E1 3761.562,E2 3761.562} C_VEL
LIN {X 0,Y 98.099,Z 1213.597,A -85,B 0,C 180,E1 3755.107,E2 3755.107} C_VEL
LIN {X 0,Y 81.07,Z 1218.953,A -85,B 0,C 180,E1 3745.721,E2 3745.721} C_VEL
LIN {X 0,Y 66.848,Z 1222.57,A -85,B 0,C 180,E1 3732.303,E2 3732.303} C_VEL
LIN {X 0,Y 57.182,Z 1224.675,A -85,B 0,C 180,E1 3713.713,E2 3713.713} C_VEL
LIN {X 0,Y 53.796,Z 1225.323,A -85,B 0,C 180,E1 3695.332,E2 3695.332} C_VEL
LIN {X 0,Y 54.753,Z 1225.213,A -85,B 0,C 180,E1 3676.268,E2 3676.268} C_VEL
LIN {X 0,Y 60.859,Z 1223.932,A -85,B 0,C 180,E1 3657.17,E2 3657.17} C_VEL
LIN {X 0,Y 72.841,Z 1221.201,A -85,B 0,C 180,E1 3640.98,E2 3640.98} C_VEL
LIN {X 0,Y 88.495,Z 1216.835,A -85,B 0,C 180,E1 3629.547,E2 3629.547} C_VEL
LIN {X 0,Y 105.544,Z 1210.955,A -85,B 0,C 180,E1 3621.819,E2 3621.819} C_VEL
LIN {X 0,Y 124.764,Z 1202.963,A -85,B 0,C 180,E1 3615.919,E2 3615.919} C_VEL
LIN {X 0,Y 143.023,Z 1193.901,A -85,B 0,C 180,E1 3611.848,E2 3611.848} C_VEL
LIN {X 0,Y 160.849,Z 1183.356,A -85,B 0,C 180,E1 3608.76,E2 3608.76} C_VEL
LIN {X 0,Y 178.057,Z 1171.484,A -85,B 0,C 180,E1 3606.337,E2 3606.337} C_VEL
LIN {X 0,Y 194.537,Z 1158.346,A -85,B 0,C 180,E1 3604.39,E2 3604.39} C_VEL
LIN {X 0,Y 204.669,Z 1149.158,A -85,B 0,C 180,E1 3603.323,E2 3603.323} C_VEL
LIN {X 0,Y 188.112,Z 1164.807,A -85,B 0,C 180,E1 3602.247,E2 3602.247} C_VEL
LIN {X 0,Y 169.984,Z 1179.778,A -85,B 0,C 180,E1 3600.721,E2 3600.721} C_VEL
LIN {X 0,Y 152.011,Z 1192.715,A -85,B 0,C 180,E1 3598.723,E2 3598.723} C_VEL
LIN {X 0,Y 132.342,Z 1204.969,A -85,B 0,C 180,E1 3595.746,E2 3595.746} C_VEL
LIN {X 0,Y 111.778,Z 1216.082,A -85,B 0,C 180,E1 3591.254,E2 3591.254} C_VEL
LIN {X 0,Y 93.134,Z 1224.89,A -85,B 0,C 180,E1 3585.056,E2 3585.056} C_VEL
LIN {X 0,Y 75,Z 1232.406,A -85,B 0,C 180,E1 3575.028,E2 3575.028} C_VEL
LIN {X 0,Y 60.46,Z 1238.102,A -85,B 0,C 180,E1 3559.527,E2 3559.527} C_VEL
LIN {X 0,Y 52.303,Z 1242.065,A -85,B 0,C 180,E1 3537.309,E2 3537.309} C_VEL
LIN {X 0,Y 51.625,Z 1242.707,A -85,B 0,C 180,E1 3531.316,E2 3531.316} C_VEL
LIN {X 0,Y 50.57,Z 1243.161,A -85,B 0,C 180,E1 3525.651,E2 3525.651} C_VEL
LIN {X 0,Y 47.802,Z 1243.142,A -85,B 0,C 180,E1 3517.509,E2 3517.509} C_VEL
LIN {X 0,Y 44.125,Z 1242.519,A -85,B 0,C 180,E1 3503.681,E2 3503.681} C_VEL
LIN {X 0,Y 44.834,Z 1240.708,A -85,B 0,C 180,E1 3479.142,E2 3479.142} C_VEL
LIN {X 0,Y 55.105,Z 1236.678,A -85,B 0,C 180,E1 3454.225,E2 3454.225} C_VEL
LIN {X 0,Y 71.845,Z 1230.861,A -85,B 0,C 180,E1 3438.86,E2 3438.86} C_VEL
LIN {X 0,Y 91.321,Z 1223.335,A -85,B 0,C 180,E1 3429.814,E2 3429.814} C_VEL
LIN {X 0,Y 111.296,Z 1214.264,A -85,B 0,C 180,E1 3424.313,E2 3424.313} C_VEL
LIN {X 0,Y 131.985,Z 1203.365,A -85,B 0,C 180,E1 3420.607,E2 3420.607} C_VEL
LIN {X 0,Y 151.047,Z 1191.776,A -85,B 0,C 180,E1 3418.217,E2 3418.217} C_VEL
LIN {X 0,Y 169.278,Z 1178.89,A -85,B 0,C 180,E1 3416.546,E2 3416.546} C_VEL
LIN {X 0,Y 176.173,Z 1173.54,A -85,B 0,C 180,E1 3416.005,E2 3416.005} C_VEL
LIN {X 0,Y 157.92,Z 1185.746,A -85,B 0,C 180,E1 3413.722,E2 3413.722} C_VEL
LIN {X 0,Y 139.731,Z 1196.132,A -85,B 0,C 180,E1 3410.91,E2 3410.91} C_VEL
LIN {X 0,Y 120.536,Z 1205.268,A -85,B 0,C 180,E1 3407.057,E2 3407.057} C_VEL
LIN {X 0,Y 102.001,Z 1212.563,A -85,B 0,C 180,E1 3401.953,E2 3401.953} C_VEL
LIN {X 0,Y 83.929,Z 1218.416,A -85,B 0,C 180,E1 3394.603,E2 3394.603} C_VEL
LIN {X 0,Y 67.223,Z 1222.711,A -85,B 0,C 180,E1 3383.432,E2 3383.432} C_VEL
LIN {X 0,Y 53.9,Z 1225.381,A -85,B 0,C 180,E1 3366.412,E2 3366.412} C_VEL
LIN {X 0,Y 46.926,Z 1226.611,A -85,B 0,C 180,E1 3344.814,E2 3344.814} C_VEL
LIN {X 0,Y 45.954,Z 1226.721,A -85,B 0,C 180,E1 3323.755,E2 3323.755} C_VEL
LIN {X 0,Y 50.024,Z 1226.094,A -85,B 0,C 180,E1 3302.632,E2 3302.632} C_VEL
LIN {X 0,Y 61.177,Z 1224.026,A -85,B 0,C 180,E1 3282.655,E2 3282.655} C_VEL
LIN {X 0,Y 76.831,Z 1220.439,A -85,B 0,C 180,E1 3269.321,E2 3269.321} C_VEL
LIN {X 0,Y 94.984,Z 1215.098,A -85,B 0,C 180,E1 3260.473,E2 3260.473} C_VEL
LIN {X 0,Y 113.631,Z 1208.249,A -85,B 0,C 180,E1 3254.562,E2 3254.562} C_VEL
LIN {X 0,Y 133.089,Z 1199.591,A -85,B 0,C 180,E1 3250.221,E2 3250.221} C_VEL
LIN {X 0,Y 152.119,Z 1189.468,A -85,B 0,C 180,E1 3247.036,E2 3247.036} C_VEL
LIN {X 0,Y 170.516,Z 1177.753,A -85,B 0,C 180,E1 3244.585,E2 3244.585} C_VEL
LIN {X 0,Y 175.882,Z 1173.969,A -85,B 0,C 180,E1 3243.957,E2 3243.957} C_VEL
LIN {X 0,Y 157.11,Z 1187.787,A -85,B 0,C 180,E1 3242.395,E2 3242.395} C_VEL
LIN {X 0,Y 137.977,Z 1200.055,A -85,B 0,C 180,E1 3240.225,E2 3240.225} C_VEL
LIN {X 0,Y 118.133,Z 1210.976,A -85,B 0,C 180,E1 3237.075,E2 3237.075} C_VEL
LIN {X 0,Y 97.871,Z 1220.546,A -85,B 0,C 180,E1 3232.275,E2 3232.275} C_VEL
LIN {X 0,Y 77.815,Z 1228.708,A -85,B 0,C 180,E1 3224.505,E2 3224.505} C_VEL
LIN {X 0,Y 60.139,Z 1235.056,A -85,B 0,C 180,E1 3211.78,E2 3211.78} C_VEL
LIN {X 0,Y 47.323,Z 1239.562,A -85,B 0,C 180,E1 3190.484,E2 3190.484} C_VEL
LIN {X 0,Y 43.66,Z 1242.23,A -85,B 0,C 180,E1 3161.894,E2 3161.894} C_VEL
LIN {X 0,Y 44.993,Z 1242.822,A -85,B 0,C 180,E1 3149.604,E2 3149.604} C_VEL
LIN {X 0,Y 44.125,Z 1242.519,A -85,B 0,C 180,E1 3143.681,E2 3143.681} C_VEL
LIN {X 0,Y 42.697,Z 1241.903,A -85,B 0,C 180,E1 3134.398,E2 3134.398} C_VEL
LIN {X 0,Y 40.415,Z 1239.971,A -85,B 0,C 180,E1 3117.048,E2 3117.048} C_VEL
LIN {X 0,Y 41.833,Z 1238.053,A -85,B 0,C 180,E1 3101.705,E2 3101.705} C_VEL
LIN {X 0,Y 43.887,Z 1237.27,A -85,B 0,C 180,E1 3096.486,E2 3096.486} C_VEL
LIN {X 0,Y 60.8,Z 1232.182,A -85,B 0,C 180,E1 3077.487,E2 3077.487} C_VEL
LIN {X 0,Y 80.684,Z 1225.484,A -85,B 0,C 180,E1 3067.539,E2 3067.539} C_VEL
LIN {X 0,Y 101.038,Z 1217.32,A -85,B 0,C 180,E1 3061.893,E2 3061.893} C_VEL
LIN {X 0,Y 121.027,Z 1207.826,A -85,B 0,C 180,E1 3058.385,E2 3058.385} C_VEL
LIN {X 0,Y 141.575,Z 1196.463,A -85,B 0,C 180,E1 3055.949,E2 3055.949} C_VEL
LIN {X 0,Y 147.453,Z 1192.835,A -85,B 0,C 180,E1 3055.381,E2 3055.381} C_VEL
LIN {X 0,Y 128.085,Z 1202.707,A -85,B 0,C 180,E1 3052.462,E2 3052.462} C_VEL
LIN {X 0,Y 108.169,Z 1210.989,A -85,B 0,C 180,E1 3048.457,E2 3048.457} C_VEL
LIN {X 0,Y 88.927,Z 1217.477,A -85,B 0,C 180,E1 3042.877,E2 3042.877} C_VEL
LIN {X 0,Y 69.977,Z 1222.543,A -85,B 0,C 180,E1 3034.176,E2 3034.176} C_VEL
LIN {X 0,Y 53.366,Z 1225.904,A -85,B 0,C 180,E1 3020.188,E2 3020.188} C_VEL
LIN {X 0,Y 41.909,Z 1227.62,A -85,B 0,C 180,E1 2998.499,E2 2998.499} C_VEL
LIN {X 0,Y 37.905,Z 1228.18,A -85,B 0,C 180,E1 2971.511,E2 2971.511} C_VEL
LIN {X 0,Y 41.141,Z 1227.746,A -85,B 0,C 180,E1 2944.059,E2 2944.059} C_VEL
LIN {X 0,Y 51.376,Z 1226.284,A -85,B 0,C 180,E1 2922.31,E2 2922.31} C_VEL
LIN {X 0,Y 67.507,Z 1223.133,A -85,B 0,C 180,E1 2907.296,E2 2907.296} C_VEL
LIN {X 0,Y 87.112,Z 1218.103,A -85,B 0,C 180,E1 2897.706,E2 2897.706} C_VEL
LIN {X 0,Y 106.279,Z 1211.843,A -85,B 0,C 180,E1 2891.933,E2 2891.933} C_VEL
LIN {X 0,Y 126.595,Z 1203.489,A -85,B 0,C 180,E1 2887.717,E2 2887.717} C_VEL
LIN {X 0,Y 145.487,Z 1194.062,A -85,B 0,C 180,E1 2884.807,E2 2884.807} C_VEL
LIN {X 0,Y 147.144,Z 1193.17,A -85,B 0,C 180,E1 2884.568,E2 2884.568} C_VEL
LIN {X 0,Y 127.092,Z 1204.835,A -85,B 0,C 180,E1 2882.427,E2 2882.427} C_VEL
LIN {X 0,Y 105.994,Z 1215.195,A -85,B 0,C 180,E1 2879.117,E2 2879.117} C_VEL
LIN {X 0,Y 85.038,Z 1223.885,A -85,B 0,C 180,E1 2873.927,E2 2873.927} C_VEL
LIN {X 0,Y 65.121,Z 1230.89,A -85,B 0,C 180,E1 2865.298,E2 2865.298} C_VEL
LIN {X 0,Y 47.579,Z 1236.239,A -85,B 0,C 180,E1 2849.494,E2 2849.494} C_VEL
LIN {X 0,Y 37.003,Z 1239.631,A -85,B 0,C 180,E1 2822.711,E2 2822.711} C_VEL
LIN {X 0,Y 36.719,Z 1241.35,A -85,B 0,C 180,E1 2791.56,E2 2791.56} C_VEL
LIN {X 0,Y 36.956,Z 1241.408,A -85,B 0,C 180,E1 2790,E2 2790} C_VEL
LIN {X 0,Y 36.744,Z 1239.739,A -85,B 0,C 180,E1 2758.869,E2 2758.869} C_VEL
LIN {X 0,Y 43.887,Z 1237.27,A -85,B 0,C 180,E1 2736.486,E2 2736.486} C_VEL
LIN {X 0,Y 47.855,Z 1235.803,A -85,B 0,C 180,E1 2728.345,E2 2728.345} C_VEL
LIN {X 0,Y 59.582,Z 1230.656,A -85,B 0,C 180,E1 2710.044,E2 2710.044} C_VEL
LIN {X 0,Y 64.911,Z 1228.954,A -85,B 0,C 180,E1 2706.695,E2 2706.695} C_VEL
LIN {X 0,Y 86.142,Z 1221.75,A -85,B 0,C 180,E1 2699.999,E2 2699.999} C_VEL
LIN {X 0,Y 108.241,Z 1212.678,A -85,B 0,C 180,E1 2696.029,E2 2696.029} C_VEL
LIN {X 0,Y 118.487,Z 1207.869,A -85,B 0,C 180,E1 2694.695,E2 2694.695} C_VEL
LIN {X 0,Y 98.24,Z 1215.377,A -85,B 0,C 180,E1 2690.824,E2 2690.824} C_VEL
LIN {X 0,Y 78.585,Z 1221.191,A -85,B 0,C 180,E1 2685.226,E2 2685.226} C_VEL
LIN {X 0,Y 59.143,Z 1225.519,A -85,B 0,C 180,E1 2675.908,E2 2675.908} C_VEL
LIN {X 0,Y 42.2,Z 1228.181,A -85,B 0,C 180,E1 2659.303,E2 2659.303} C_VEL
LIN {X 0,Y 31.924,Z 1229.397,A -85,B 0,C 180,E1 2632.076,E2 2632.076} C_VEL
LIN {X 0,Y 30.332,Z 1229.503,A -85,B 0,C 180,E1 2600.514,E2 2600.514} C_VEL
LIN {X 0,Y 36.698,Z 1228.887,A -85,B 0,C 180,E1 2571.199,E2 2571.199} C_VEL
LIN {X 0,Y 51.749,Z 1226.829,A -85,B 0,C 180,E1 2549.607,E2 2549.607} C_VEL
LIN {X 0,Y 70.414,Z 1223.249,A -85,B 0,C 180,E1 2537.946,E2 2537.946} C_VEL
LIN {X 0,Y 90.648,Z 1217.909,A -85,B 0,C 180,E1 2530.993,E2 2530.993} C_VEL
LIN {X 0,Y 110.705,Z 1211.058,A -85,B 0,C 180,E1 2526.557,E2 2526.557} C_VEL
LIN {X 0,Y 118.223,Z 1208.131,A -85,B 0,C 180,E1 2525.217,E2 2525.217} C_VEL
LIN {X 0,Y 97.055,Z 1217.568,A -85,B 0,C 180,E1 2522.205,E2 2522.205} C_VEL
LIN {X 0,Y 75.088,Z 1225.727,A -85,B 0,C 180,E1 2517.032,E2 2517.032} C_VEL
LIN {X 0,Y 54.242,Z 1232.083,A -85,B 0,C 180,E1 2507.672,E2 2507.672} C_VEL
LIN {X 0,Y 36.446,Z 1236.564,A -85,B 0,C 180,E1 2488.259,E2 2488.259} C_VEL
LIN {X 0,Y 27.764,Z 1239.326,A -85,B 0,C 180,E1 2448.911,E2 2448.911} C_VEL
LIN {X 0,Y 28.812,Z 1239.97,A -85,B 0,C 180,E1 2430,E2 2430} C_VEL
LIN {X 0,Y 30.344,Z 1238.148,A -85,B 0,C 180,E1 2388.776,E2 2388.776} C_VEL
LIN {X 0,Y 44.732,Z 1234.498,A -85,B 0,C 180,E1 2360.157,E2 2360.157} C_VEL
LIN {X 0,Y 64.911,Z 1228.954,A -85,B 0,C 180,E1 2346.695,E2 2346.695} C_VEL
LIN {X 0,Y 68.977,Z 1227.549,A -85,B 0,C 180,E1 2344.14,E2 2344.14} C_VEL
LIN {X 0,Y 78.55,Z 1223.222,A -85,B 0,C 180,E1 2336.383,E2 2336.383} C_VEL
LIN {X 0,Y 82.387,Z 1221.735,A -85,B 0,C 180,E1 2335.094,E2 2335.094} C_VEL
LIN {X 0,Y 89.197,Z 1219.302,A -85,B 0,C 180,E1 2333.894,E2 2333.894} C_VEL
LIN {X 0,Y 68.397,Z 1224.576,A -85,B 0,C 180,E1 2328.35,E2 2328.35} C_VEL
LIN {X 0,Y 48.337,Z 1228.178,A -85,B 0,C 180,E1 2318.559,E2 2318.559} C_VEL
LIN {X 0,Y 30.283,Z 1230.31,A -85,B 0,C 180,E1 2296.583,E2 2296.583} C_VEL
LIN {X 0,Y 22.428,Z 1230.904,A -85,B 0,C 180,E1 2260.272,E2 2260.272} C_VEL
LIN {X 0,Y 25.685,Z 1230.746,A -85,B 0,C 180,E1 2216.977,E2 2216.977} C_VEL
LIN {X 0,Y 39.079,Z 1229.439,A -85,B 0,C 180,E1 2189.555,E2 2189.555} C_VEL
LIN {X 0,Y 59.081,Z 1226.466,A -85,B 0,C 180,E1 2175.289,E2 2175.289} C_VEL
LIN {X 0,Y 79.803,Z 1221.98,A -85,B 0,C 180,E1 2168.202,E2 2168.202} C_VEL
LIN {X 0,Y 89.097,Z 1219.429,A -85,B 0,C 180,E1 2165.996,E2 2165.996} C_VEL
LIN {X 0,Y 67.012,Z 1226.765,A -85,B 0,C 180,E1 2161.505,E2 2161.505} C_VEL
LIN {X 0,Y 45.293,Z 1232.412,A -85,B 0,C 180,E1 2152.391,E2 2152.391} C_VEL
LIN {X 0,Y 25.67,Z 1236.503,A -85,B 0,C 180,E1 2126.959,E2 2126.959} C_VEL
LIN {X 0,Y 20.184,Z 1238.394,A -85,B 0,C 180,E1 2075.686,E2 2075.686} C_VEL
LIN {X 0,Y 20.637,Z 1238.528,A -85,B 0,C 180,E1 2070,E2 2070} C_VEL
LIN {X 0,Y 24.699,Z 1236.679,A -85,B 0,C 180,E1 2015.943,E2 2015.943} C_VEL
LIN {X 0,Y 42.599,Z 1233.007,A -85,B 0,C 180,E1 1989.454,E2 1989.454} C_VEL
LIN {X 0,Y 64.997,Z 1227.322,A -85,B 0,C 180,E1 1979.064,E2 1979.064} C_VEL
LIN {X 0,Y 82.387,Z 1221.735,A -85,B 0,C 180,E1 1975.094,E2 1975.094} C_VEL
LIN {X 0,Y 81.016,Z 1222.034,A -85,B 0,C 180,E1 1974.411,E2 1974.411} C_VEL
LIN {X 0,Y 73.44,Z 1224.064,A -85,B 0,C 180,E1 1973.69,E2 1973.69} C_VEL
LIN {X 0,Y 57.405,Z 1228.111,A -85,B 0,C 180,E1 1974.056,E2 1974.056} C_VEL
LIN {X 0,Y 47.895,Z 1230.246,A -85,B 0,C 180,E1 1975.874,E2 1975.874} C_VEL
LIN {X 0,Y 26.319,Z 1234.435,A -85,B 0,C 180,E1 1988.997,E2 1988.997} C_VEL
LIN {X 0,Y 12.051,Z 1236.719,A -85,B 0,C 180,E1 2045.858,E2 2045.858} C_VEL
LIN {X 0,Y 12.446,Z 1237.082,A -85,B 0,C 180,E1 2070,E2 2070} C_VEL
LIN {X 0,Y 21.339,Z 1235.163,A -85,B 0,C 180,E1 2143.677,E2 2143.677} C_VEL
LIN {X 0,Y 43.726,Z 1231.195,A -85,B 0,C 180,E1 2162.624,E2 2162.624} C_VEL
LIN {X 0,Y 58.95,Z 1227.608,A -85,B 0,C 180,E1 2167.157,E2 2167.157} C_VEL
LIN {X 0,Y 37.651,Z 1230.664,A -85,B 0,C 180,E1 2177.062,E2 2177.062} C_VEL
LIN {X 0,Y 20.91,Z 1232.034,A -85,B 0,C 180,E1 2200.09,E2 2200.09} C_VEL
LIN {X 0,Y 14.378,Z 1232.331,A -85,B 0,C 180,E1 2257.994,E2 2257.994} C_VEL
LIN {X 0,Y 23.909,Z 1231.807,A -85,B 0,C 180,E1 2306.76,E2 2306.76} C_VEL
LIN {X 0,Y 43.213,Z 1229.976,A -85,B 0,C 180,E1 2326.351,E2 2326.351} C_VEL
LIN {X 0,Y 59.107,Z 1227.535,A -85,B 0,C 180,E1 2332.932,E2 2332.932} C_VEL
LIN {X 0,Y 47.895,Z 1230.246,A -85,B 0,C 180,E1 2335.874,E2 2335.874} C_VEL
LIN {X 0,Y 41.402,Z 1231.514,A -85,B 0,C 180,E1 2336.996,E2 2336.996} C_VEL
LIN {X 0,Y 32.557,Z 1232.575,A -85,B 0,C 180,E1 2335.495,E2 2335.495} C_VEL
LIN {X 0,Y 14.407,Z 1233.556,A -85,B 0,C 180,E1 2316.234,E2 2316.234} C_VEL
LIN {X 0,Y 13.404,Z 1233.575,A -85,B 0,C 180,E1 2313.885,E2 2313.885} C_VEL
LIN {X 0,Y 7.465,Z 1233.692,A -85,B 0,C 180,E1 2217.608,E2 2217.608} C_VEL
LIN {X 0,Y 22.549,Z 1233.126,A -85,B 0,C 180,E1 2172.71,E2 2172.71} C_VEL
LIN {X 0,Y 26.68,Z 1232.931,A -85,B 0,C 180,E1 2169.441,E2 2169.441} C_VEL
LIN {X 0,Y 5.686,Z 1235.26,A -85,B 0,C 180,E1 2131.546,E2 2131.546} C_VEL
LIN {X 0,Y 4.228,Z 1235.632,A -85,B 0,C 180,E1 2070,E2 2070} C_VEL
LIN {X 0,Y 21.149,Z 1233.604,A -85,B 0,C 180,E1 1973.103,E2 1973.103} C_VEL
LIN {X 0,Y 26.687,Z 1232.89,A -85,B 0,C 180,E1 1970.331,E2 1970.331} C_VEL
LIN {X 0,Y 13.404,Z 1233.575,A -85,B 0,C 180,E1 1953.885,E2 1953.885} C_VEL
LIN {X 0,Y 11.742,Z 1235.575,A -85,B 0,C 180,E1 1949.059,E2 1949.059} C_VEL
LIN {X 0,Y 11.742,Z 1319.5,A -85,B 0,C 180,E1 1949.059,E2 1949.059} C_VEL
LIN {X 0,Y 11.742,Z 1319.5,A -85,B 0,C 180,E1 1949.059,E2 1949.059}

QRS_NEXT_CUT()

QRS_NEXT()
QRS_HOME()

END
